TYPE HmiControl :
STRUCT
	counter		: UDINT;
END_STRUCT
END_TYPE

(* stored: Version 1.1.0.1, ProductVersion 3.1.4020.12
   DUT HmiControl: Id {277bad6a-a1eb-42d6-a5ae-8450c2594cd2} *)
